// Mitsubishi GX Works2 project: exercicio set reset   PLC: Q03UDV

PROGRAM MAIN
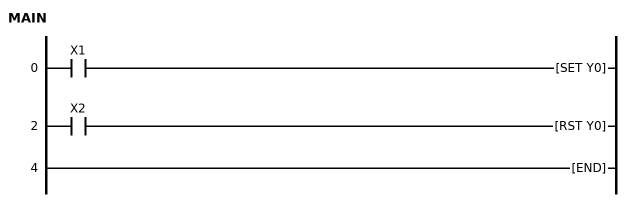
0     LD      X1
      SET     Y0
2     LD      X2
      RST     Y0
4     END
END_PROGRAM
